FUNCTION_BLOCK TCFB (* Timing contract function block *)
  (* Standard: 61499-2 *)
  (* Version 1.0, 2018-10-23, Duc Do Tran, OFFIS e.V. *)
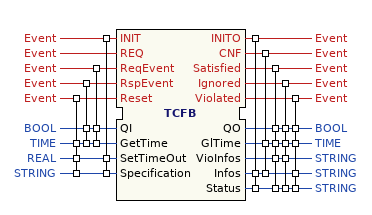
  EVENT_INPUT
    INIT WITH Specification, SetTimeOut;
    REQ;
    ReqEvent WITH QI, GetTime;
    RspEvent WITH QI, GetTime;
    Reset WITH Specification, SetTimeOut, GetTime;
  END_EVENT
  EVENT_OUTPUT
    INITO WITH Status, Infos;
    CNF WITH Infos, GlTime;
    Satisfied WITH QO, Status, VioInfos, GlTime;
    Ignored WITH Status, QO, VioInfos, GlTime;
    Violated WITH QO, Status, Infos, GlTime;
  END_EVENT
  VAR_INPUT
    QI : BOOL := 1;
    GetTime : TIME := 0;
    SetTimeOut : REAL := 60;
    Specification : STRING;
  END_VAR
  VAR_OUTPUT
    QO : BOOL;
    GlTime : TIME;
    VioInfos : STRING;
    Infos : STRING;
    Status : STRING;
  END_VAR
  VAR
    Pass : BOOL; (* Internal Variable *)
    ipo : STRING := |; (* Internal Variable *)
    ExceptHdl : BOOL; (* Internal Variable *)
    nsec : STRING := ns; (* Internal Variable *)
    usec : STRING := us; (* Internal Variable *)
    msec : STRING := ms; (* Internal Variable *)
    sec : STRING := s; (* Internal Variable *)
    ob : STRING := [; (* open bracket *)
    cb : STRING := ]; (* close bracket *)
    ep : STRING := #; (* exclamation point *)
    P1 : STRING; (* Internal Variable *)
    P2 : STRING; (* Internal Variable *)
    P3 : STRING; (* Internal Variable *)
    P4 : STRING; (* Internal Variable *)
    beginP : STRING := e(; (* Internal Variable *)
    endP : STRING := ); (* Internal Variable *)
    in : STRING := |=; (* Internal Variable *)
    eq : STRING := =; (* Internal Variable *)
    qst : STRING := ->; (* Internal Variable *)
    dcm : STRING := ;; (* Internal Variable *)
    dbp : STRING := :; (* Internal Variable *)
    AE : BOOL; (* Internal Variable *)
    eExt : STRING := }; (* Internal Variable *)
    bExt : STRING := {; (* Internal Variable *)
    P5 : STRING; (* Internal Variable *)
    ExtCmd : STRING; (* Internal Variable *)
    tt : REAL; (* Internal Variable *)
    tunit : STRING; (* Internal Variable *)
    Pattern : STRING; (* Internal Variable *)
    ReqArr : ARRAY [0..999] OF TIME; (* Internal Variable *)
    PosV : ARRAY [0..999] OF INT; (* Internal Variable *)
    NumEV : INT; (* Internal Variable *)
    MaxNum : REAL; (* Internal Variable *)
    MinNum : REAL; (* Internal Variable *)
    Occurr : STRING := Occurrence; (* Internal Variable *)
    React : STRING := Reaction; (* Internal Variable *)
    Age : STRING := Age; (* Internal Variable *)
    Causal : STRING := Causality; (* Internal Variable *)
    Class : STRING := ::; (* Internal Variable *)
    RspNum : INT; (* Internal Variable *)
    Done : BOOL; (* Internal Variable *)
    bd : BOOL; (* Internal Variable *)
    Fulfilled : BOOL; (* Internal Variable *)
    RspArr : ARRAY [0..999] OF TIME; (* Internal Variable *)
    ConstraintType : STRING; (* Internal Variable *)
    LastPosV : INT; (* Internal Variable *)
    CountReq : INT := 0; (* Internal Variable *)
    CountRsp : INT; (* Internal Variable *)
    i : INT; (* Internal Variable *)
    j : INT; (* Internal Variable *)
    MaxNum1 : REAL; (* Internal Variable *)
    MinNum1 : REAL; (* Internal Variable *)
    beginP1 : STRING := q(; (* Internal Variable *)
    ReqNum1 : INT; (* Internal Variable *)
    RspNum1 : INT; (* Internal Variable *)
    Num : SINT; (* Internal Variable *)
    ReactCase : USINT; (* Internal Variable *)
    VNum : INT; (* Internal Variable *)
    CountReq1 : UINT; (* Internal Variable *)
    CountRsp1 : UINT; (* Internal Variable *)
    Temp : ARRAY [0..999] OF INT; (* Internal Variable *)
    LastReq : TIME; (* Internal Variable *)
    TempStr : STRING; (* Internal Variable *)
    flag : BOOL; (* Internal Variable *)
    TempStr1 : STRING; (* Internal Variable *)
    FirstTime : TIME; (* Internal Variable *)
    ReqTout : BOOL; (* Internal Variable *)
    RspTout : BOOL; (* Internal Variable *)
    t : ARRAY [0..999] OF LREAL; (* Internal Variable *)
    cma : STRING := ,; (* Internal Variable *)
    LastTime : TIME; (* Internal Variable *)
    Te : REAL; (* Internal Variable *)
    CurrTime : TIME; (* Internal Variable *)
    IgnAct : BOOL; (* Internal Variable *)
    StrVar : STRING; (* Internal Variable *)
    Timeout : BOOL; (* Internal Variable *)
    TimeoutVal : REAL; (* Internal Variable *)
    beginTimeout : TIME; (* Internal Variable *)
    ErrorCode : USINT; (* Internal Variable *)
  END_VAR
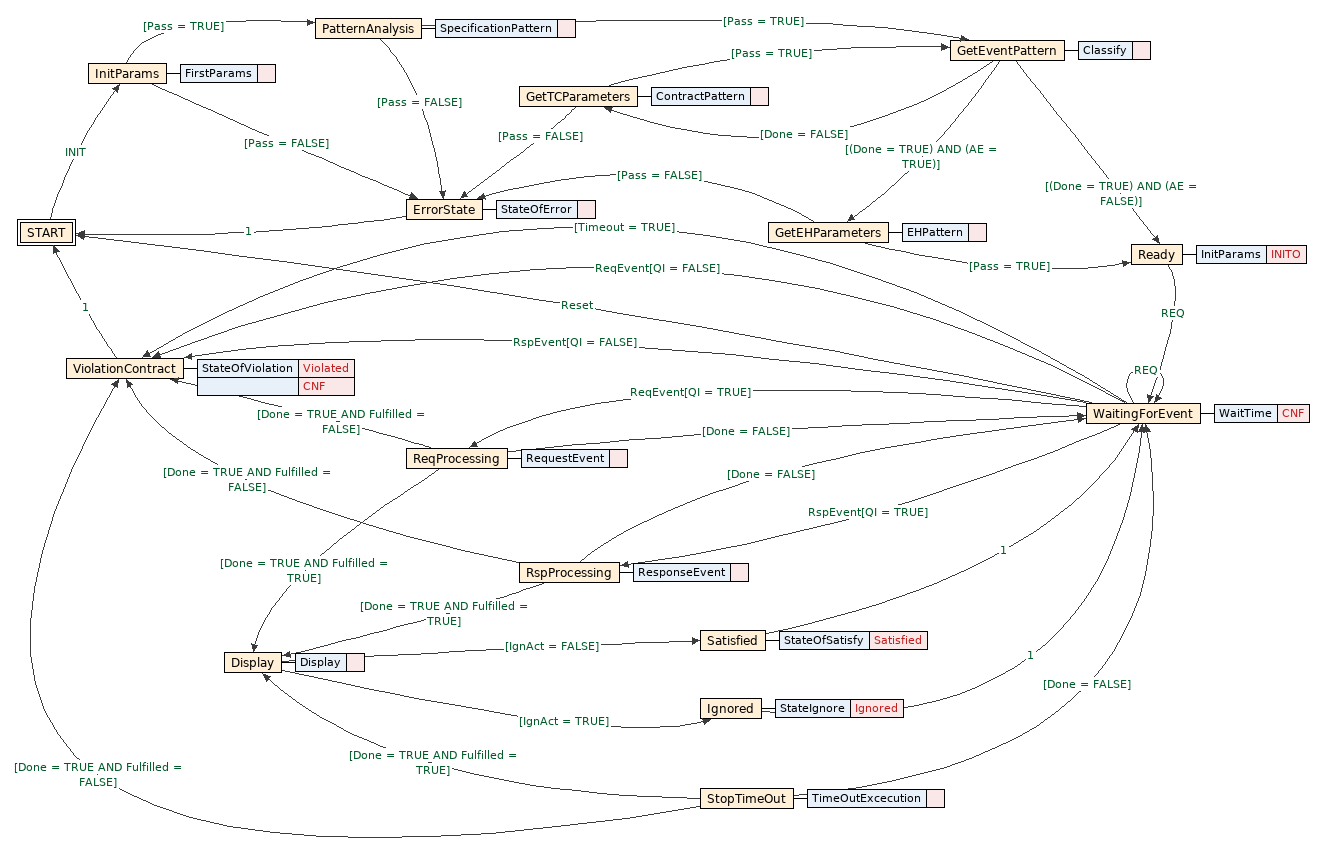
  EC_STATES
    START; (* Initial State *)
    PatternAnalysis : SpecificationPattern;
    ReqProcessing : RequestEvent;
    GetTCParameters : ContractPattern;
    GetEventPattern : Classify;
    WaitingForEvent : WaitTime -> CNF;
    RspProcessing : ResponseEvent;
    ErrorState : StateOfError;
    Display : Display;
    ViolationContract : StateOfViolation -> Violated, -> CNF;
    Ready : InitParams -> INITO;
    InitParams : FirstParams;
    GetEHParameters : EHPattern;
    StopTimeOut : TimeOutExcecution;
    Satisfied : StateOfSatisfy -> Satisfied;
    Ignored : StateIgnore -> Ignored;
  END_STATES
  EC_TRANSITIONS
    GetTCParameters TO GetEventPattern := [Pass = TRUE];
    PatternAnalysis TO ErrorState := [Pass = FALSE];
    GetTCParameters TO ErrorState := [Pass = FALSE];
    ReqProcessing TO ViolationContract := [Done = TRUE AND Fulfilled = FALSE];
    RspProcessing TO ViolationContract := [Done = TRUE AND Fulfilled = FALSE];
    GetEventPattern TO Ready := [(Done = TRUE) AND (AE = FALSE)];
    ViolationContract TO START := 1;
    ErrorState TO START := 1;
    GetEventPattern TO GetTCParameters := [Done = FALSE];
    START TO InitParams := INIT;
    InitParams TO PatternAnalysis := [Pass = TRUE];
    GetEHParameters TO ErrorState := [Pass = FALSE];
    InitParams TO ErrorState := [Pass = FALSE];
    StopTimeOut TO Display := [Done = TRUE AND Fulfilled = TRUE];
    Display TO Satisfied := [IgnAct = FALSE];
    Display TO Ignored := [IgnAct = TRUE];
    ReqProcessing TO Display := [Done = TRUE AND Fulfilled = TRUE];
    RspProcessing TO Display := [Done = TRUE AND Fulfilled = TRUE];
    WaitingForEvent TO ViolationContract := [Timeout = TRUE];
    WaitingForEvent TO START := Reset;
    WaitingForEvent TO ReqProcessing := ReqEvent[QI = TRUE];
    WaitingForEvent TO RspProcessing := RspEvent[QI = TRUE];
    WaitingForEvent TO ViolationContract := RspEvent[QI = FALSE];
    WaitingForEvent TO ViolationContract := ReqEvent[QI = FALSE];
    Satisfied TO WaitingForEvent := 1;
    Ignored TO WaitingForEvent := 1;
    RspProcessing TO WaitingForEvent := [Done =  FALSE];
    ReqProcessing TO WaitingForEvent := [Done =  FALSE];
    StopTimeOut TO ViolationContract := [Done = TRUE AND Fulfilled = FALSE];
    WaitingForEvent TO WaitingForEvent := REQ;
    PatternAnalysis TO GetEventPattern := [Pass = TRUE];
    GetEHParameters TO Ready := [Pass = TRUE];
    GetEventPattern TO GetEHParameters := [(Done = TRUE) AND (AE = TRUE)];
    StopTimeOut TO WaitingForEvent := [Done =  FALSE];
    Ready TO WaitingForEvent := REQ;
  END_TRANSITIONS
  ALGORITHM SpecificationPattern IN ST: (* new algorithm *)
IF (LEN(Specification) > 0) THEN //Occurrence:: | Occurrence::e(t|=[a;b]ms) | Reaction::q(i|=[39.6,40.4]]s)?e(i|=[19.8,20.2]s)
	IF (LEN(LEFT(Specification, FIND(Specification,Class))) > 0) THEN
		StrVar := LEFT(Specification, FIND(Specification,Class));
		ConstraintType := LEFT(StrVar, LINT_TO_ULINT(LEN(StrVar) - 1)); // Occurrence| Reaction | Age
		P1 := RIGHT(Specification, LINT_TO_ULINT(LEN(Specification) - LEN(ConstraintType) - LEN(Class))); // P1 : e(p=5ms:j=1ms) or e(i|=[a;b]ms) or e(p=5ms:j=1ms)# Exception
		IF (ConstraintType = Occurr) THEN
			IF((LEFT(P1, LINT_TO_ULINT(2)) = beginP )AND (RIGHT(P1, LINT_TO_ULINT(1)) = endP)) THEN
				Num := 1;
				ReactCase := 0;
			ELSE
				Pass := FALSE;
				ErrorCode := 2;
				//Infos := "Invalid syntax of specification :: check again syntax e(...)";
			END_IF;
		ELSIF ((ConstraintType = React) OR (ConstraintType = Age))  THEN //P1 = q?e(i|=[a;b]ms)[#][{...|...}]Or P1 = q(i|=[a;b]ms)?e(i|=[a;b]ms)[#][{...|...}]
			StrVar := LEFT(P1, FIND(P1,qst));
			P2 := LEFT(StrVar, LINT_TO_ULINT(LEN(StrVar) - 1)); //q | q(i|=[a;b]ms)
			P1 := RIGHT(P1, LINT_TO_ULINT(LEN(P1) - LEN(P2) - LEN(qst))); //e(i|=[a;b]ms)[#][{...|...}]
			IF(P2 = "q") THEN
				Num := 1;
				ReactCase := 1;
		 	ELSE
		 		IF (RIGHT(P2, LINT_TO_ULINT(1)) = endP) AND (LEFT(P2, LINT_TO_ULINT(2)) = beginP1) THEN
			 		ReactCase := 2;
				 	Num := 2;
				ELSE
					Pass := FALSE;
					ErrorCode := 2;
					//Infos := "Invalid syntax of specification :: check again syntax q(...)";
				END_IF;
			END_IF;

			IF ((LEFT(P1, LINT_TO_ULINT(2)) = beginP) AND (LEN(LEFT(P1, FIND(P1,endP))) > 0))  THEN
				IF (RIGHT(P1, LINT_TO_ULINT(1)) <> endP) THEN
					IF (LEN(LEFT(P1, FIND(P1,ep))) >0) THEN
						StrVar := LEFT(P1, FIND(P1,ep));	//....#EXT
						P3 := LEFT(StrVar, LINT_TO_ULINT(LEN(StrVar) - 1)); //e(i|=[a;b]ms)
						IF (RIGHT(P3,LINT_TO_ULINT(1)) = endP) THEN
					 		ExtCmd := RIGHT(P1, LINT_TO_ULINT(LEN(P1) - LEN(P3) -1));//[#][{...|...}]
					 		P1 := P3;
					 		IF (LEN(ExtCmd) >= 1) THEN
						 		IF (LEN(LEFT(ExtCmd, FIND(ExtCmd,bExt))) > 0) THEN
						 			StrVar := LEFT(ExtCmd, FIND(ExtCmd,bExt));
						 			P3 := LEFT(StrVar, LINT_TO_ULINT(LEN(StrVar) - 1));
						 			RspNum := STRING_TO_INT(P3);
						 			ExtCmd := RIGHT(ExtCmd, LINT_TO_ULINT(LEN(ExtCmd) - LEN(P3)));
						 			IF (LEN(ExtCmd) >= 5) THEN
										AE := TRUE;
									ELSE
										Pass := FALSE;
										Infos := "Error:: The exception handling command is failed!!!";
									END_IF;
								ELSE
									ExceptHdl := TRUE;
									VioInfos := ExtCmd;
									RspNum := STRING_TO_INT(ExtCmd);
								END_IF;
							ELSE
								Pass := FALSE;
								Infos := "Error:: The exception handling command is failed!!!";
							END_IF;
						ELSE
							Pass := FALSE;
							Infos := "Invalid syntax of specification :: check again syntax e(...)";
						END_IF;
					ELSE
						IF (LEN(LEFT(P1, FIND(P1,bExt))) > 0) THEN
							StrVar := LEFT(P1, FIND(P1,bExt));
							P3 := LEFT(StrVar, LINT_TO_ULINT(LEN(StrVar) - 1));
							IF (RIGHT(P3,LINT_TO_ULINT(1)) = endP) THEN
								ExtCmd := RIGHT(P1, LINT_TO_ULINT(LEN(P1) - LEN(P3)));
								P1 := P3;
								IF (LEN(ExtCmd) >= 5) THEN
									AE := TRUE;
								ELSE
									Pass := FALSE;
									Infos := "Error:: The exception handling command is failed!!!";
								END_IF;
							ELSE
								Pass := FALSE;
								Infos := "Invalid syntax of specification :: check syntax e(...) or needs with '#'";
							END_IF;
						ELSE
							Pass := FALSE;
							Infos := "Error:: that needs begin with '#' or '{'";
						END_IF;
					END_IF;
				END_IF;
			 ELSE
				Pass := FALSE;
				Infos := "Invalid syntax of specification :: check again syntax e(...)";
	 		END_IF;
		ELSIF(ConstraintType = Causal) THEN

		ELSE
			Pass := FALSE;
			Infos := ConstraintType; //(i|=[39.6,40.4]]s)?e(i|=[19.8,20.2]s)
			//Infos := "Invalid syntax of specification :: invalid keyword of contract ";
		END_IF;
	ELSE
		Pass := FALSE;
		Infos := "Invalid syntax of specification :: missing or invalid symbol of class '::' ";
	END_IF;
ELSE
		Pass := FALSE;
		Infos := "Invalid syntax of specification :: empty specification";
END_IF;
  END_ALGORITHM
  ALGORITHM RequestEvent IN ST: (* new algorithm *)
IF (GetTime = 0) THEN
	LastReq := NOW_MONOTONIC();
ELSE
	LastReq := GetTime;
END_IF;
GlTime := LastReq;

IF (ConstraintType = Occurr) THEN
	Done := TRUE;
	IF (bd = TRUE) THEN
		FirstTime := LastReq;
		bd := FALSE;
		TimeoutVal := MaxNum;
	ELSE
		IF (TIME_IN_S_TO_LREAL(LastReq - FirstTime) >= MinNum) AND (TIME_IN_S_TO_LREAL(LastReq - FirstTime) <= MaxNum) THEN
			FirstTime :=  LastReq;
		ELSE
			Fulfilled := FALSE;
			Infos := "Request event is not fulfilled for the requirement of period time.";
		END_IF;
	END_IF;
	beginTimeout  :=  LastReq;
ELSIF (ConstraintType = React) THEN
	flag := FALSE;
	IF (ReqTout = TRUE) THEN
		CountRsp := 0;
		ReqTout := FALSE;
		TimeoutVal := MaxNum;
		beginTimeout  :=  LastReq;
		IF (VNum > 0) THEN
			CountReq := CountReq + 1;
		END_IF;
		IF (bd = TRUE) THEN
			FirstTime := LastReq;
			bd := FALSE;
		ELSE
			IF (ReactCase = 2) THEN
				IF (TIME_IN_S_TO_LREAL(LastReq - FirstTime)< MinNum1) THEN
					Fulfilled := FALSE;
					Done := TRUE;
					VNum := VNum + 1;
					Infos := "The requested event occurs earlier than the required!!!";
				ELSIF (TIME_IN_S_TO_LREAL(LastReq - FirstTime) > MaxNum1) THEN
					Fulfilled := FALSE;
					Done := TRUE;
					VNum := VNum + 1;
					Infos := "The requested event occurs later than the required!!!";
				ELSE
					FirstTime := LastReq;
				END_IF;
			END_IF;
		END_IF;
	ELSE //the response event is not fulfilled.
		Fulfilled := FALSE;
		Done := TRUE;
		VNum := VNum + 1;

		/*Infos := "Too many request event.";
		VNum := VNum + 1;
		IF (TIME_IN_S_TO_LREAL(LastReq - FirstTime)< MinNum1) THEN
			Fulfilled := FALSE;
			Done := TRUE;
			Infos := "The requested event occurs earlier than the required!!!";
		ELSIF (TIME_IN_S_TO_LREAL(LastReq - FirstTime) > MaxNum1) THEN
			Fulfilled := FALSE;
			Done := TRUE;
			Infos := "The requested event occurs later than the required!!!";
		ELSE
			CountRsp := 0;
			ReqTout := FALSE;
			TimeoutVal := MaxNum;
			beginTimeout  :=  LastReq;
			IF (VNum > 0) THEN
				CountReq := CountReq + 1;
			END_IF;
		END_IF;
		*

		IF (ExceptHdl = TRUE) THEN
			IF (ReactCase = 2) THEN
				IF (TIME_IN_S_TO_LREAL(LastReq - FirstTime)< MinNum1) THEN
					Fulfilled := FALSE;
					Done := TRUE;
					VNum := VNum + 1;
					Infos := "The requested event occurs earlier than the required!!!";
				ELSIF (TIME_IN_S_TO_LREAL(LastReq - FirstTime) > MaxNum1) THEN
					Fulfilled := FALSE;
					Done := TRUE;
					VNum := VNum + 1;
					Infos := "The requested event occurs later than the required!!!";
				ELSE
					VNum := VNum + 1;
					CountRsp := 0;
					ReqTout := FALSE;
					TimeoutVal := MaxNum;
					beginTimeout  :=  LastReq;
					IF (VNum > 0) THEN
						CountReq := CountReq + 1;
					END_IF;
				END_IF;
			ELSE
				Fulfilled := FALSE;
				Done := TRUE;
				VNum := VNum + 1;
			END_IF;
		ELSE
			Fulfilled := FALSE;
			Done := TRUE;
			VNum := VNum + 1;
			Infos := "Too many request event.";
		END_IF;	*/
	END_IF;
	//----------------------------------------------------------------------ooo
ELSIF (ConstraintType = Age) THEN
		CountReq := CountReq + 1;
		ReqArr[CountReq] := LastReq;
		TimeoutVal := MaxNum;
		beginTimeout := LastReq;
		/*IF (ReqTout = TRUE) THEN
		 	ReqTout := FALSE;
			beginTimeout  :=  LastReq;
			IF (bd = TRUE) THEN
				FirstTime := LastReq;
				bd := FALSE;
				CountRsp :=0;
				Done := TRUE;
			ELSE
				Done := TRUE;
				IF (VNum > 0) THEN
					CountReq := CountReq + 1;
				ELSE
					CountReq := 1;
					VNum := 0;
				END_IF;
				IF (ReactCase = 2) THEN
					IF (TIME_IN_S_TO_LREAL(LastReq - FirstTime)< MinNum1) THEN
						Fulfilled := FALSE;
						VNum := VNum + 1;
						Status := "The requested event occurs earlier than the required!!!";
					ELSIF (TIME_IN_S_TO_LREAL(LastReq - FirstTime) > MaxNum1) THEN
						Fulfilled := FALSE;
						VNum := VNum + 1;
						Status := "The requested event occurs later than the required!!!";
					ELSE
						TimeoutVal := MaxNum1 - MinNum;
						FirstTime := LastReq;
					END_IF;
				ELSE
					TimeoutVal := SetTimeOut - MinNum;
					FirstTime := LastReq;
				END_IF;

				IF (Fulfilled = TRUE) THEN
					j := 0;
					LastPosV := 0;
					IF (CountRsp > 0) THEN
						TempStr := "Set of backward times: ";
						FOR i := 1 TO CountRsp DO
							t[i] :=TIME_IN_S_TO_LREAL(LastReq - RspArr[i]);
							IF (t[i] > MaxNum) THEN
								IF(RspArr[i] <> 0) THEN
									LastPosV := i;
								END_IF;
							ELSIF (t[i] >= MinNum) AND (t[i] <= MaxNum) THEN
								j := j + 1;
								LastPosV := i;
							ELSE
								//EXIT;
							END_IF;
							TempStr1 := CONCAT(LREAL_TO_STRING(t[i]),ipo);
							TempStr := CONCAT(TempStr,TempStr1);
						END_FOR;
						Infos := TempStr;
					END_IF;
					IF (RspNum <> j) THEN
						Fulfilled := FALSE;
						IF (ExceptHdl = TRUE) THEN
							VNum := VNum + 1;
							IF (VNum <= NumEV) THEN
								Fulfilled := TRUE;
								PosV[VNum] :=CountReq;
								IgnAct := TRUE;
							ELSE
								Infos := "Number of violation is exceed the allowed times of exception handling";
								VNum := VNum + 1;
							END_IF;
						ELSE
							Infos := "Number of response times do not meet requirement";
							VNum := VNum + 1;
						END_IF;
					END_IF;

					IF (Fulfilled = TRUE) THEN
						IF (LastPosV > 0) THEN
							CountRsp := CountRsp - LastPosV;
							IF (CountRsp > 0) THEN
								FOR i := 1 TO CountRsp DO
									RspArr[i] := RspArr[i +LastPosV];
									RspArr[i +LastPosV] := 0;
								END_FOR;
							ELSE
								CountRsp := 0;
								FOR i := 1 TO LastPosV DO
									RspArr[i] := 0;
								END_FOR;
							END_IF;
						END_IF;
					END_IF;
				END_IF;
			END_IF;
		ELSE
			Fulfilled := FALSE;
			Done := TRUE;
			VNum := VNum + 1;
			Infos := "Too many request event.";
		END_IF; */


///=================================
		/*IF (bd = FALSE) THEN
			IF (ReactCase = 2) THEN
				TimeoutVal := MaxNum1;
			ELSE
				TimeoutVal := MaxNum;//SetTimeOut - Te;
			END_IF;
			TempStr := "Reaction time Te = ";
			TempStr1 := REAL_TO_STRING(Te);
			Infos := CONCAT(TempStr,TempStr1);
		ELSE
			Infos := "Waiting for first response event.";
		END_IF;	*/
///================================
ELSE
	Done := FALSE;
END_IF;
  END_ALGORITHM
  ALGORITHM ResponseEvent IN ST: (* new algorithm *)
CurrTime := NOW_MONOTONIC();
IF(ConstraintType <> Occurr) THEN
	Te := TIME_IN_S_TO_LREAL(CurrTime - LastReq);
	Infos := "";
	IF (ConstraintType = React) THEN
		IF(bd = FALSE) THEN
			IF (Te >= MinNum) AND (Te <= MaxNum) THEN
				CountRsp := CountRsp + 1;
				IF (CountRsp = RspNum) THEN
					Done := TRUE;
					ReqTout := TRUE;
					beginTimeout := CurrTime;
					IF (ReactCase = 2) THEN
						TimeoutVal := MaxNum1 - Te;
					ELSE
						TimeoutVal := SetTimeOut  - Te;
					END_IF;
				ELSIF  (CountRsp < RspNum) THEN
					TempStr := "Number of response event: ";
					TempStr1 := INT_TO_STRING(CountRsp);
					 Infos := CONCAT(TempStr,TempStr1);
				ELSE
					IF (ExceptHdl = TRUE) THEN
						IF (flag = FALSE) THEN
							flag := TRUE;
							VNum := VNum + 1;
							IF (VNum <= NumEV) THEN
								PosV[VNum] :=CountReq;
								VioInfos := INT_TO_STRING(CountReq);
								IgnAct := TRUE;
								TempStr := INT_TO_STRING(RspNum);
								TempStr1 := INT_TO_STRING(CountRsp);
								TempStr1 := CONCAT(TempStr1,ipo);
								TempStr := CONCAT(TempStr1,TempStr);
								TempStr1 := "Satisfied RspEv | Reqiured RspEv: ";
								Infos := CONCAT(TempStr1,TempStr);
								Done := TRUE;
							ELSE
								Fulfilled := FALSE;
								VNum := VNum + 1;
								Infos := "Number of violation is exceed the allowed times of exception handling";
								Done := TRUE;
							END_IF;
						ELSE
							TempStr := INT_TO_STRING(RspNum);
							TempStr1 := INT_TO_STRING(CountRsp);
							TempStr1 := CONCAT(TempStr1,ipo);
							TempStr := CONCAT(TempStr1,TempStr);
							TempStr1 := "Satisfied RspEv | Reqiured RspEv: ";
							Infos := CONCAT(TempStr1,TempStr);
						END_IF;
					ELSE
						Fulfilled := FALSE;
						VNum := VNum + 1;
						Infos := "Number of response event is exceed the desired times";
						Done := TRUE;
					END_IF;
				END_IF;
			ELSIF (Te > MaxNum) THEN
				IF (CountRsp >= RspNum) THEN
					TempStr := INT_TO_STRING(RspNum);
					TempStr1 := INT_TO_STRING(CountRsp);
					TempStr1 := CONCAT(TempStr1,ipo);
					TempStr := CONCAT(TempStr1,TempStr);
					TempStr1 := "Satisfied RspEv | Reqiured RspEv: ";
					Infos := CONCAT(TempStr1,TempStr);
				END_IF;
			ELSE
				Infos := "Waiting for next response event.";
				beginTimeout := LastTime;
				TimeoutVal := MaxNum - Te;
			END_IF;
		ELSE
			Infos := "Waiting for first request event.";
		END_IF;
	ELSIF (ConstraintType = Age) THEN
		j :=0;
		IF (CountReq > 0) THEN
			TempStr := "Set of backward times: ";
			FOR i := 1 TO CountReq DO
				t[i] :=TIME_IN_S_TO_LREAL(CurrTime - ReqArr[i]);
				IF (t[i] >= MinNum) AND (t[i] <= MaxNum) THEN
					j := j + 1;
					TempStr1 := CONCAT(LREAL_TO_STRING(t[i]),ipo);
					TempStr := CONCAT(TempStr,TempStr1);
				END_IF;
			END_FOR;
			Infos := TempStr;
			IF ( j <> 1) THEN
				Fulfilled := FALSE;
				Done := TRUE;
				IF (ExceptHdl = TRUE) THEN
					VNum := VNum + 1;
					IF (VNum <= NumEV) THEN
						Fulfilled := TRUE;
						PosV[VNum] :=CountReq;
						IgnAct := TRUE;
					ELSE
						Infos := "Number of violation is exceed the allowed times of exception handling";
						VNum := VNum + 1;
					END_IF;
				ELSE
					Infos := "Number of response times do not meet requirement";
					VNum := VNum + 1;
				END_IF;
			ELSE
				CountReq := 0;
				Done := TRUE;
				beginTimeout := CurrTime;
				Te := SetTimeOut  -  TIME_IN_S_TO_LREAL(CurrTime - LastReq);
				IF (ReactCase = 2) THEN
					TimeoutVal := MaxNum1 - Te;
				ELSE
					TimeoutVal:= SetTimeOut  -  Te;
				END_IF;
			END_IF;
		ELSE
			Fulfilled := FALSE;
			Infos := "No request!";
		END_IF;

	ELSE

	END_IF;
END_IF;
  END_ALGORITHM
  ALGORITHM Classify IN ST: (* new algorithm *)
IF (Num = 2)  THEN
	Pattern  := RIGHT(P2, LINT_TO_ULINT(LEN(P2) - LEN(beginP1))); // P1 : q(i|=[a;b]ms)
ELSIF (Num = 1) THEN
	Pattern := RIGHT(P1, LINT_TO_ULINT(LEN(P1) - LEN(beginP)));
ELSE
	Done := TRUE;
END_IF;
  END_ALGORITHM
  ALGORITHM InitParams IN ST: (* new algorithm *)
beginTimeout := NOW_MONOTONIC();
LastTime := NOW_MONOTONIC();
CurrTime := NOW_MONOTONIC();
bd := TRUE;
Timeout := FALSE;
IF (CountRsp > 0) THEN
	FOR i := 1 TO CountRsp DO
		RspArr[i] := 0;
	END_FOR;
END_IF;
ReqTout := TRUE;
VNum := 0;
IF (ConstraintType = Age) THEN
	CountReq :=0;
ELSE
	CountReq :=1;
END_IF;
IF (ReqNum1 > 0) THEN
	NumEV := ReqNum1 - RspNum1;
END_IF;
Fulfilled := TRUE;
  END_ALGORITHM
  ALGORITHM StateOfSatisfy IN ST: (* new algorithm *)
IF (ConstraintType = Age) THEN
	//TempStr1 := "||";
	//TempStr := LREAL_TO_STRING(TIME_IN_S_TO_LREAL(LastReq - RspArr[1]));
	//TempStr1 := CONCAT(TempStr,TempStr1);
	//Status:= CONCAT(TempStr1,LREAL_TO_STRING(TIME_IN_S_TO_LREAL(LastReq - RspArr[2])));
	Status := "Contract is satisfied.";
ELSE
	TempStr := ": Contract is satisfied.";
	TempStr1 := "Te = :";
	TempStr1 := CONCAT(TempStr1,REAL_TO_STRING(Te));
	Status:= CONCAT(TempStr1,TempStr);
END_IF;
  END_ALGORITHM
  ALGORITHM StateOfViolation IN ST: (* new algorithm *)
QO := FALSE;
IF (QI = FALSE) THEN
	Status := "Invalid status";
	Infos := "Not allowed QI = 0.";
ELSE
	Status := "Contract is violated.";
	TempStr := "Number of violation: ";
	TempStr1 := INT_TO_STRING(VNum+1);
	Infos := CONCAT(TempStr,TempStr1);
	IF (Timeout = TRUE) THEN
		VioInfos := "Time out";
	ELSE
		TempStr := "Mearsured Time: ";
		TempStr1 := "Te = ";
		TempStr1 := CONCAT(TempStr1,REAL_TO_STRING(Te));
		VioInfos := CONCAT(TempStr,TempStr1);
	END_IF;
END_IF;
  END_ALGORITHM
  ALGORITHM StateOfError IN ST: (* new algorithm *)
QO := FALSE;
Status := P1;//"An error has occurred!";
  END_ALGORITHM
  ALGORITHM ContractPattern IN ST: (* new algorithm *)
IF (LEN(LEFT(Pattern, FIND(Pattern,endP))) > 0 ) THEN
	StrVar := LEFT(Pattern, FIND(Pattern,endP));			// P1 :  i|=[a;b]ms
	P5 := LEFT(StrVar, LINT_TO_ULINT(LEN(StrVar) - 1));
	StrVar := LEFT(P5, FIND(P5,in));
	IF (LEFT(StrVar, LINT_TO_ULINT(LEN(StrVar) - 1)) = "i") THEN
		P3 := RIGHT(P5, LINT_TO_ULINT(LEN(P5) - LEN(in) - 1));//P3 := "[a;b]ms"
		IF (LEFT(P3, FIND(P3, nsec)) <> 0) THEN
			tunit := nsec;
			tt := 0.000000001;
		ELSIF (LEFT(P3, FIND(P3, usec)) <> 0) THEN
			tunit := usec;
			tt := 0.000001;
		ELSIF (LEFT(P3, FIND(P3, msec)) <> 0) THEN
			tunit := msec;
			tt := 0.001;
		ELSIF (LEFT(P3, FIND(P3, sec)) <> 0) THEN
			tunit := sec;
			tt := 1;
		ELSE
			Pass := FALSE;
			Infos := "Error :: invalid unit  of time";
		END_IF;
	ELSE
		Pass := FALSE;
		Infos := "Error :: invalid variable of specification for time interval";
	END_IF;

	IF (Pass = TRUE) THEN
		StrVar :=  LEFT(P3, FIND(P3, tunit));//P2 := "[a;b]"
		P3 := LEFT(StrVar, LINT_TO_ULINT(LEN(StrVar) - 1));
		IF ((LEFT(P3, LINT_TO_ULINT(1)) = ob) AND (RIGHT(P3, LINT_TO_ULINT(1)) = cb)) THEN
			IF (LEN(LEFT(P3, FIND(P3,cma))) > 0) THEN
				StrVar := LEFT(P3, FIND(P3,cma));  //P3 := "[a"
				P4 := LEFT(StrVar, LINT_TO_ULINT(LEN(StrVar) - 1));
				P5 := RIGHT(P3, LINT_TO_ULINT(LEN(P3) - LEN(P4) - 1));//P2 := "b]"
				IF (LEN(RIGHT(P5, LINT_TO_ULINT(LEN(P5) - 1))) > 0) THEN
					P4 := RIGHT(P4, LINT_TO_ULINT(LEN(P4) - 1)); //P3 := "a"
					StrVar := LEFT(P5, FIND(P5,cb));
					P5 := LEFT(StrVar, LINT_TO_ULINT(LEN(StrVar) - 1));
					MinNum :=  STRING_TO_REAL(P4)*tt;
					MaxNum :=  STRING_TO_REAL(P5)*tt;
					IF (MaxNum <= MinNum) THEN
						Pass := FALSE;
						Infos := "Error :: check again the interval values  [min,max]?';'";
					ELSE
						IF (Num = 2) THEN
							MinNum1 :=  MinNum;
							MaxNum1 :=  MaxNum;
						END_IF;
					END_IF;
				ELSE
					Pass := FALSE;
					Infos := "Error :: empty or unvalid timing data ';'";
				END_IF;
			ELSE
				Pass := FALSE;
				Infos := "Error :: missing ',' between two values";
			END_IF;
		ELSE
			Pass := FALSE;
			Infos := "Invalid syntax of specification :: missing or unvalid symbol of interval [...,...]";
		END_IF;
	END_IF;
ELSE
	Pass := FALSE;
	Infos := "Error :: unkown variable of specification";
END_IF;
Num := Num - 1;
  END_ALGORITHM
  ALGORITHM FirstParams IN ST: (* new algorithm *)
Infos := "";
Status := "";
VioInfos := "";
Pass := TRUE;
Done := FALSE;
AE := FALSE;
ExceptHdl := FALSE;
ReqNum1 := 0;
RspNum1 := 0;
RspNum := 1;
//ReqNum := 1;
ReactCase := 0;
IF (SetTimeOut <=0) THEN
	Pass := FALSE;
	Infos := "Invalid timeout value";
ELSE
	TimeoutVal := SetTimeOut;
END_IF;
  END_ALGORITHM
  ALGORITHM WaitTime IN ST: (* new algorithm *)
Fulfilled := TRUE;
Done := FALSE;
Timeout := FALSE;
IgnAct := FALSE;
IF (TIME_IN_S_TO_LREAL(NOW_MONOTONIC() - beginTimeout) > TimeoutVal) AND (bd = FALSE) THEN
	Timeout := TRUE;
END_IF;
  END_ALGORITHM
  ALGORITHM EHPattern IN ST: (* new algorithm *)
 ExceptHdl := TRUE;
IF ((LEFT(ExtCmd,  LINT_TO_ULINT(1)) = bExt)  AND (RIGHT(ExtCmd,  LINT_TO_ULINT(1)) = eExt)) THEN
	IF (ConstraintType = Occurr) THEN
		Pass := FALSE;
		Infos := "Error:: This command does not required for this case";
	ELSE
		 IF (LEN(LEFT(ExtCmd, FIND(ExtCmd,ipo))) > 0) THEN
			StrVar := LEFT(ExtCmd, FIND(ExtCmd,ipo));
			P4 := LEFT(StrVar, LINT_TO_ULINT(LEN(StrVar) - 1));//P4 := "{a"
			P5 := RIGHT(ExtCmd, LINT_TO_ULINT(LEN(ExtCmd) - LEN(P4) - 1));//P2 := "b}"
			IF ((LEN(P4) > 1) AND (LEN(P5) > 1)) THEN
				P4 := RIGHT(P4, LINT_TO_ULINT(LEN(P4) - 1)); //P4 := "a"
				StrVar := LEFT(P5, FIND(P5,eExt));
				P5 := LEFT(StrVar, LINT_TO_ULINT(LEN(StrVar) - 1));
				RspNum1 :=  STRING_TO_INT(P4);
				ReqNum1 :=  STRING_TO_INT(P5);
			ELSE
				Pass := FALSE;
				Infos := "Error:: Missing input or/and output value for exception handling";
			END_IF;
		ELSE
			Pass := FALSE;
			Infos := "Error:: Missing symbol '|'";
		END_IF;
	END_IF;
ELSE
	IF (LEN(LEFT(Specification, FIND(Specification,ep))) = 0) THEN
		Pass := FALSE;
		Infos := "Error:: Check again syntax {...|...}";
	END_IF;
END_IF;
  END_ALGORITHM
  ALGORITHM TimeOutExcecution IN ST: (* new algorithm *)
beginTimeout := NOW_MONOTONIC();
Fulfilled := FALSE;
Done := TRUE;
/*
IF (ReqTout = TRUE) THEN
	Infos := "Timout for request event!!!";
	VNum := VNum + 1;
ELSE
	IF (ConstraintType = React) THEN
		IF (ExceptHdl = TRUE) AND (flag = FALSE) THEN
			VNum := VNum + 1;
			IF (VNum <= NumEV) THEN
				Fulfilled := TRUE;
				ReqTout := TRUE;
				PosV[VNum] :=CountReq;
				VioInfos := INT_TO_STRING(CountReq);
				TempStr := INT_TO_STRING(RspNum);
				TempStr1 := INT_TO_STRING(CountRsp);
				TempStr1 := CONCAT(TempStr1,ipo);
				TempStr := CONCAT(TempStr1,TempStr);
				TempStr1 := "Satisfied RspEv | Reqiured RspEv: ";
				Infos := CONCAT(TempStr1,TempStr);
				flag := TRUE;
				IgnAct := TRUE;
				IF (ReactCase = 2) THEN
					TimeoutVal := MaxNum1 -  TIME_IN_S_TO_LREAL(beginTimeout - LastReq);
				ELSE
					TimeoutVal := SetTimeOut -  TIME_IN_S_TO_LREAL(beginTimeout - LastReq);
				END_IF;
			ELSE
				Fulfilled := FALSE;
				Infos := "Number of violation is exceed the allowed times of exception handling";
				VNum := VNum + 1;
			END_IF;
		ELSE
			Done := TRUE;
			Fulfilled := FALSE;
			Infos := "Timeout.";
		END_IF;
	ELSE
		IF (ConstraintType = Age) THEN
			ReqTout := TRUE;
			IF (ReactCase = 2) THEN
				TimeoutVal := MaxNum1 - TIME_IN_S_TO_LREAL(beginTimeout - LastReq);
			ELSE
				TimeoutVal := SetTimeOut  - TIME_IN_S_TO_LREAL(beginTimeout - LastReq);
			END_IF;
			TempStr := INT_TO_STRING(RspNum);
			TempStr1 := INT_TO_STRING(CountRsp);
			TempStr1 := CONCAT(TempStr1,ipo);
			Infos := CONCAT(TempStr1,TempStr);
		ELSE

		END_IF;
	END_IF;
END_IF;*/
//TempStr := INT_TO_STRING(RspNum);
//TempStr1 := INT_TO_STRING(CountRsp);
//TempStr1 := CONCAT(TempStr1,ipo);
//Infos := CONCAT(TempStr1,TempStr);
  END_ALGORITHM
  ALGORITHM Display IN ST: (* new algorithm *)
QO := TRUE;
IF (VNum > 0) THEN
	IF (CountReq > ReqNum1) THEN
		CountReq := ReqNum1;
		VioInfos := "";
		TempStr := "List of violation position: ";
		FOR i :=1 TO VNum DO
			Temp[i] := PosV[i] - 1;
			IF (Temp[i] < 0) THEN
				PosV[i] := 0;
			 	EXIT;
			 END_IF;
		END_FOR;
		IF (Temp[1]  = 0) THEN
			VNum := VNum - 1;
			IF (VNum > 0) THEN
				FOR j :=1 TO VNum DO
					PosV[j] := Temp[j+1];
					TempStr1 := CONCAT(INT_TO_STRING(PosV[j]),ipo);
					TempStr := CONCAT(TempStr,TempStr1);
				END_FOR;
			ELSE
				VNum := 0;
				CountReq := 1;
				TempStr := "";
			END_IF;
		ELSE
			FOR j :=1 TO VNum DO
				PosV[j] := Temp[j];
				TempStr1 := CONCAT(INT_TO_STRING(PosV[j]),ipo);
				TempStr := CONCAT(TempStr,TempStr1);
			END_FOR;
		END_IF;
	ELSE
		VioInfos := "";
		TempStr := "List of violation position of contract: ";
		FOR j :=1 TO VNum DO
			TempStr1 := CONCAT(INT_TO_STRING(PosV[j]),ipo);
			TempStr := CONCAT(TempStr,TempStr1);
		END_FOR;
	END_IF;
	VioInfos := TempStr;
ELSE
	VNum := 0;
	CountReq := 1;
	VioInfos := "No errors";
END_IF;
  END_ALGORITHM
  ALGORITHM StateIgnore IN ST: (* new algorithm *)
IF (ConstraintType = Age) THEN
	Status := ": Contract is ignored by exception handling.";
ELSE
	TempStr := ": Contract is ignored by exception handling.";
	TempStr1 := "Te = :";
	TempStr1 := CONCAT(TempStr1,REAL_TO_STRING(Te));
	Status:= CONCAT(TempStr1,TempStr);
END_IF;
  END_ALGORITHM
END_FUNCTION_BLOCK
